//Funzione che ritorna TRUE se almeno un modulo è in errore
FUNCTION TFPalletizerIsModuleError : bool 
VAR_INPUT
	Modules : POINTER TO TFPalletizerModules;
END_VAR
VAR
END_VAR

TFPalletizerIsModuleError := TFIsModuleError(Modules^.AX_X.Error)OR
								TFIsModuleError(Modules^.AX_Y.Error)OR
								TFIsModuleError(Modules^.AX_Z.Error)OR
								TFIsModuleError(Modules^.AX_J.Error)OR
								TFIsModuleError(Modules^.Pinza.Error);

END_FUNCTION

(* stored: Version 1.1.0.1, ProductVersion 3.1.4024.11
   POU TFPalletizerIsModuleError: Id {7edb5307-49b9-46f3-a633-7365319a3652}, SpecialFunc None *)
